PROGRAM P_ScrewersCharts_1


VAR
    fbFileOpen   : FB_FileOpen;
    fbFileClose  : FB_FileClose;
    fbFileWrite  : FB_FileWrite;
    hFile        : UINT := 0;(* File handle *)

    sFilePath    : STRING(400); //:= 'C:\Recipe_changes\RecipeChanges.txt'
    bSave        : BOOL;(* Trigger to start the file saving *)
    bBusy        : BOOL;
    bError       : BOOL;
    nErrId       : UDINT;
    
    Step         : DWORD := 0;(* Step for state machine *)
    nIndex       : INT := 0;(* Index for array iteration *)
    sBuffer      : STRING(3000);(* Buff	er for writing to file *)
    nBytesToWrite: DINT;
    dtString     : STRING(25);
    nTotalItems  : INT := 500;(* Total items in array *)
	nZeroCountInBuffer:int;
    RisingEdge   : R_TRIG;
	bNonZeroDetected:BOOL;
	nZeroCount:INT;
	i:INT;
	nDataLength:INT;
	ColIndex: INT := 500;
	DataArray:ARRAY[0..500]OF INT;
	ftbRun:f_trig;
	
    nIndex_l: INT := 1;
    bWrite1: BOOL; 
	bWrite2: BOOL;
    nValueToWrite: INT; 
    bError1: BOOL := FALSE;
    nErrId1: UINT; 
	bhandy1:bool;
	
	lrPreviousValueTorqueSetted:LREAL;
	
	
	
	
END_VAR
VAR_INPUT
	nFileCounter :INT:=2;
END_VAR


//P10_GripperScrewer.fb2GripperScrewer1.bCycleDone1

ftbRun(clk:= P_ADS_SCREW.bScrewer1Run);
RisingEdge(CLK := ftbRun.Q );//OR P_ADS_Screw.bScrewer1Done1 OR P_ADS_Screw.bScrewer1Done2 OR P_ADS_Screw.bScrewer1NotDone1 OR ftbRun.q);
CASE Step OF
    0:
        IF RisingEdge.Q THEN
            bBusy := TRUE;
            bError := FALSE;
            nErrId := 0;
            nIndex := 0;
            sFilePath := CONCAT('C:\LastScrewingCycles\Zakrecarka_1_', INT_TO_STRING(nFileCounter));
            sFilePath := CONCAT(sFilePath, '.csv');
            nFileCounter := nFileCounter + 1;
            IF nFileCounter > 50 THEN
                nFileCounter := 1;
            END_IF
            Step := 10;
        END_IF
    10:
        // Kopiowanie wszystkich danych do DataArray
        FOR i := 0 TO 500 DO
            DataArray[i] := P_ADS_Screw.AStChartGripperScrewer1[0][2, i];
        END_FOR
        nDataLength := 500; // Ustaw pełną długość danych
        Step := 20;
    20:
        // Otwórz plik do zapisu
        fbFileOpen(sNetId := '', sPathName := sFilePath,
                   nMode := FOPEN_MODEWRITE OR FOPEN_MODETEXT,
                   ePath := PATH_GENERIC,
                   bExecute := TRUE);
        Step := 30;
    30:
        fbFileOpen(bExecute := FALSE);
        IF NOT fbFileOpen.bBusy THEN
            IF fbFileOpen.bError THEN
                nErrId := fbFileOpen.nErrId;
                bError := TRUE;
                Step := 500;
            ELSE
                hFile := fbFileOpen.hFile;
                Step := 40;
            END_IF
        END_IF
    40:
        // Zapisz dane w mniejszych porcjach (np. po 100 wierszy)
        IF nIndex <= nDataLength THEN
            sBuffer := '';
            FOR i := nIndex TO MIN(nIndex + 99, nDataLength) DO
                sBuffer := CONCAT(sBuffer, INT_TO_STRING(DataArray[i]));
				sBuffer := CONCAT(sBuffer, '$N');
            END_FOR
            nBytesToWrite := LEN(sBuffer);
            fbFileWrite(sNetId := '', hFile := hFile,
                        pWriteBuff := ADR(sBuffer),
                        cbWriteLen := nBytesToWrite,
                        bExecute := TRUE);
            Step := 50;
        ELSE
            Step := 300; // Przejdź do zamknięcia pliku po zapisaniu wszystkich danych
        END_IF
    50:
        fbFileWrite(bExecute := FALSE);
        IF NOT fbFileWrite.bBusy THEN
            IF fbFileWrite.bError THEN
                nErrId := fbFileWrite.nErrId;
                bError := TRUE;
                Step := 500;
            ELSE
                nIndex := nIndex + 100; // Przejdź do następnej porcji danych
                Step := 40;
            END_IF
        END_IF
    300:
        // Zamknij plik
        fbFileClose(sNetId := '', hFile := hFile, bExecute := TRUE);
        Step := 310;
    310:
        fbFileClose(bExecute := FALSE);
        IF NOT fbFileClose.bBusy THEN
            IF fbFileClose.bError THEN
                nErrId := fbFileClose.nErrId;
                bError := TRUE;
            END_IF
            Step := 500;
        END_IF
    500:
        // Zakończ eksport
        bBusy := FALSE;
        bSave := FALSE;
        Step := 0;
        nIndex := 0; 
END_CASE

bWrite1:=ftbRun.q;
IF bWrite1 THEN
    IF nValueToWrite >= 0 THEN
        gvl_screw.aLast50Screw1[nIndex_l] := p_ads_screw.lrGripperScrewer1TorqueCV;
        nIndex_l := nIndex_l + 1;
        IF nIndex_l > 500 THEN
            nIndex_l := 1;
        END_IF;
        bWrite1 := FALSE;
    ELSE
        bError1 := TRUE;
        nErrId1 := 1;
    END_IF;
END_IF;

IF lrPreviousValueTorqueSetted<>P_ADS_SCREW.lrGripperScrewingTightTorqueShow OR bhandy1 THEN
	for i:=1 to 501 do
		gvl_screw.a50ScrewSetted1[i]:=P_ADS_SCREW.lrGripperScrewingTightTorqueShow;
	END_FOR
	lrPreviousValueTorqueSetted:=P_ADS_SCREW.lrGripperScrewingTightTorqueShow;
END_IF;

END_PROGRAM

(* stored: Version 1.2.0.0, ProductVersion 3.1.4026.13, FileIdentifier a37d4a9979419c0bd2b1b835e7cae976c7b92e04, FileSignature 3e4d68791a22185a002dd7acfaff2cf8bb49c8eb8edbd30042d2b2e64eba9295aa665f4cc6d35427b00910d65b9bbdef325e2242de17b380408d73bb42b21f70076740b26ace3c1332354c397ff2c466e1e4aeade4ef9d62b1e1fe6477155d4f76baa8fd342a23c538da3a9bf6ba9d1d304695df20dd67d250bc2ea41f43b783b8ac501b8b43840eb1ccb61ad512d1ffca54e1dffa805c8fd8400cd20ec6622b95b5c399ba847b81a19e163470603fe499a7fd672e6d4816b40c37eb21ee829098ef2b4ff3a8204bc7ae243164aa2a62028ec747f71f6b4f4cd80e9e236fe12d4e8d149059aa31ea9188abb63a5cdc03dd6b9915454c7451099551f7a7cc9f98
   POU P_ScrewersCharts_1: Id {d2c04254-5daf-42cd-9d10-f98732e80df2}, SpecialFunc None *)
